// SIMATIC S7-200 SMART project (STEP 7-Micro/WIN SMART), CPU ST40

SYMBOL_TABLE Table 1
Start_SW         I0.0
Stop_Sw          I0.1
Memory_1         M0.0
Memory_2         M0.1
FWD              Q0.0
REV              Q0.1
OFF_Timer_1      T101
FWD_Timer        T102
OFF_Timer_2      T103
REV_Timer        T104
END_SYMBOL_TABLE

ORGANIZATION_BLOCK MAIN:OB1
TITLE=Program Comments
BEGIN
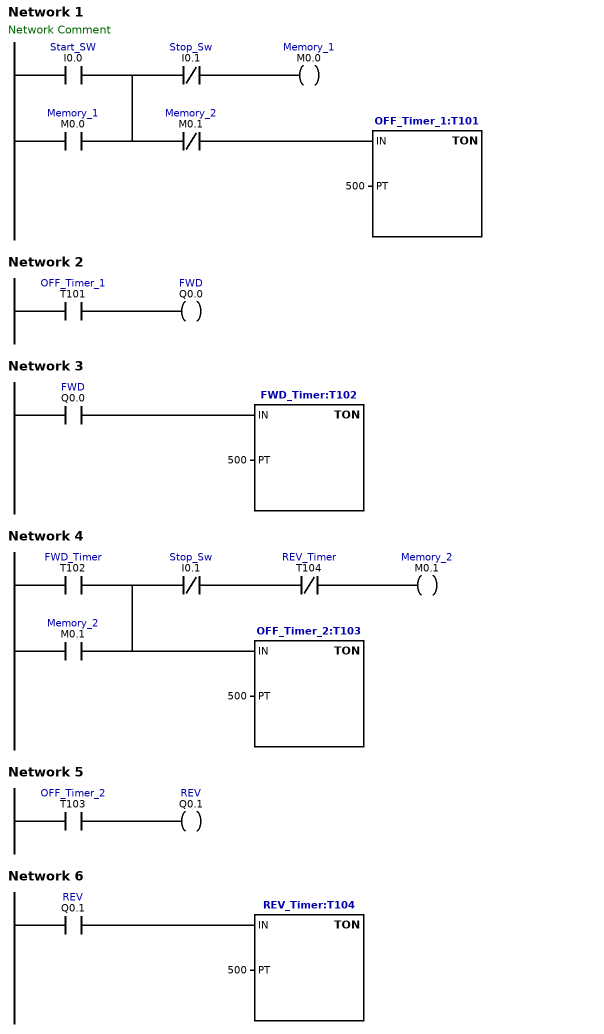
Network 1
// Network Comment
LD     Start_SW:I0.0
O      Memory_1:M0.0
LPS
AN     Stop_Sw:I0.1
=      Memory_1:M0.0
LPP
AN     Memory_2:M0.1
TON    OFF_Timer_1:T101, 500
Network 2
LD     OFF_Timer_1:T101
=      FWD:Q0.0
Network 3
LD     FWD:Q0.0
TON    FWD_Timer:T102, 500
Network 4
LD     FWD_Timer:T102
O      Memory_2:M0.1
LPS
AN     Stop_Sw:I0.1
AN     REV_Timer:T104
=      Memory_2:M0.1
LPP
TON    OFF_Timer_2:T103, 500
Network 5
LD     OFF_Timer_2:T103
=      REV:Q0.1
Network 6
LD     REV:Q0.1
TON    REV_Timer:T104, 500
END_ORGANIZATION_BLOCK
